FUNCTION_BLOCK CAR_MOVE
VAR_INPUT
END_VAR
VAR_OUTPUT
END_VAR
VAR
END_VAR

// NETWORK 1

END_FUNCTION_BLOCK

(* stored: Version 1.1.0.1
   POU CAR_MOVE: Id {477bffb7-a49c-4d89-b031-21b5e5baedba}, SpecialFunc None *)
